(* PLC project ammonium-nitrates, Generated TextualNotationConverter 1.0 *)
(* stored: creationDateTime 2025-07-30T12:00:00, modificationDateTime 2025-01-30T12:00:00 *)

FUNCTION_BLOCK ANALOG_IN
  VAR_INPUT
    Name : STRING;
    Description : STRING;
    Raw_Signal : REAL;
    PV_High : REAL;
    PV_Low : REAL;
    Scaling_Slope : REAL;
    Scaling_Offset : REAL;
    Alarm_Enable : BOOL;
  END_VAR
  VAR_OUTPUT
    PV : REAL;
    High_Alarm : BOOL;
    Low_Alarm : BOOL;
    General_Fault : BOOL;
  END_VAR

            
          
END_FUNCTION_BLOCK

FUNCTION_BLOCK BOOL_IN
  VAR_INPUT
    Name : STRING;
    Description : STRING;
    Bool_In : BOOL;
    Alarm_OnTrue : BOOL;
    Alarm_OnFalse : BOOL;
    Latch_Enable : BOOL;
    Reset_Latch : BOOL;
  END_VAR
  VAR_OUTPUT
    Bool_Out : BOOL;
    Alarm_Active : BOOL;
    Latched_Status : BOOL;
  END_VAR

            
          
END_FUNCTION_BLOCK

FUNCTION_BLOCK PID_BASIC
  VAR_INPUT
    Name : STRING;
    Description : STRING;
    AUTO : BOOL;
    PV : REAL;
    SP : REAL;
    MV_MIN : REAL;
    MV_MAX : REAL;
    X0 : REAL;
    KP : REAL;
    TR : REAL;
    TD : REAL;
    PV_High : REAL;
    PV_Low : REAL;
    Deviation_Limit : REAL;
    Inhibit : BOOL;
  END_VAR
  VAR_OUTPUT
    PV_High_Alarm : BOOL;
    PV_Low_Alarm : BOOL;
    Deviation_Alarm : BOOL;
    XOUT : REAL;
  END_VAR

            
          
END_FUNCTION_BLOCK

FUNCTION_BLOCK RATIO_CONTROL
  VAR_INPUT
    Name : STRING;
    Description : STRING;
    Auto : BOOL;
    PrimaryPV : REAL;
    SecondaryPV : REAL;
    RatioSP : REAL;
    Bias : REAL;
    TrimKp : REAL;
    TrimTi : STRING;
    MV_MIN : REAL;
    MV_MAX : REAL;
    ManOut : REAL;
    Inhibit : BOOL;
  END_VAR
  VAR_OUTPUT
    SlaveSP : REAL;
    ActiveRatio : REAL;
    RatioErr : REAL;
  END_VAR

            
          
END_FUNCTION_BLOCK

FUNCTION_BLOCK VALVE_ELECTRIC
  VAR_INPUT
    Name : STRING;
    Description : STRING;
    Control_Signal : REAL;
    Manual_Mode : BOOL;
    Manual_Position : REAL;
    Open_Limit : REAL;
    Close_Limit : REAL;
    Timeout : STRING;
    Inhibit : BOOL;
  END_VAR
  VAR_OUTPUT
    Valve_Position : REAL;
    Feedback_Pos : REAL;
    Valve_Moving : BOOL;
    Position_Error : BOOL;
    Alarm : BOOL;
  END_VAR

            
          
END_FUNCTION_BLOCK

PROGRAM Section2
  VAR
    FIC102_AcidFlow_SP_FromRatio : REAL;
    FV102_ValveCmd_Pct : REAL;
    FV101_ValveCmd_Pct : REAL;
    FT101_AmmoniaFlow_PV : REAL;
  END_VAR
  VAR
    FT-101 : ANALOG_IN;
    FT-102 : ANALOG_IN;
    LT-104 : ANALOG_IN;
    PH-105 : ANALOG_IN;
    FIC-101 : PID_BASIC;
    FIC-102 : PID_BASIC;
    TIC-103 : PID_BASIC;
    FFIC-102 : RATIO_CONTROL;
    FV-101 : VALVE_ELECTRIC;
    FV-102 : VALVE_ELECTRIC;
    VS-107 : BOOL_IN;
  END_VAR
  VAR  (* added by the conversion: wires and edge detectors of the diagram *)
    _OR1_OUT : BOOL;
  END_VAR

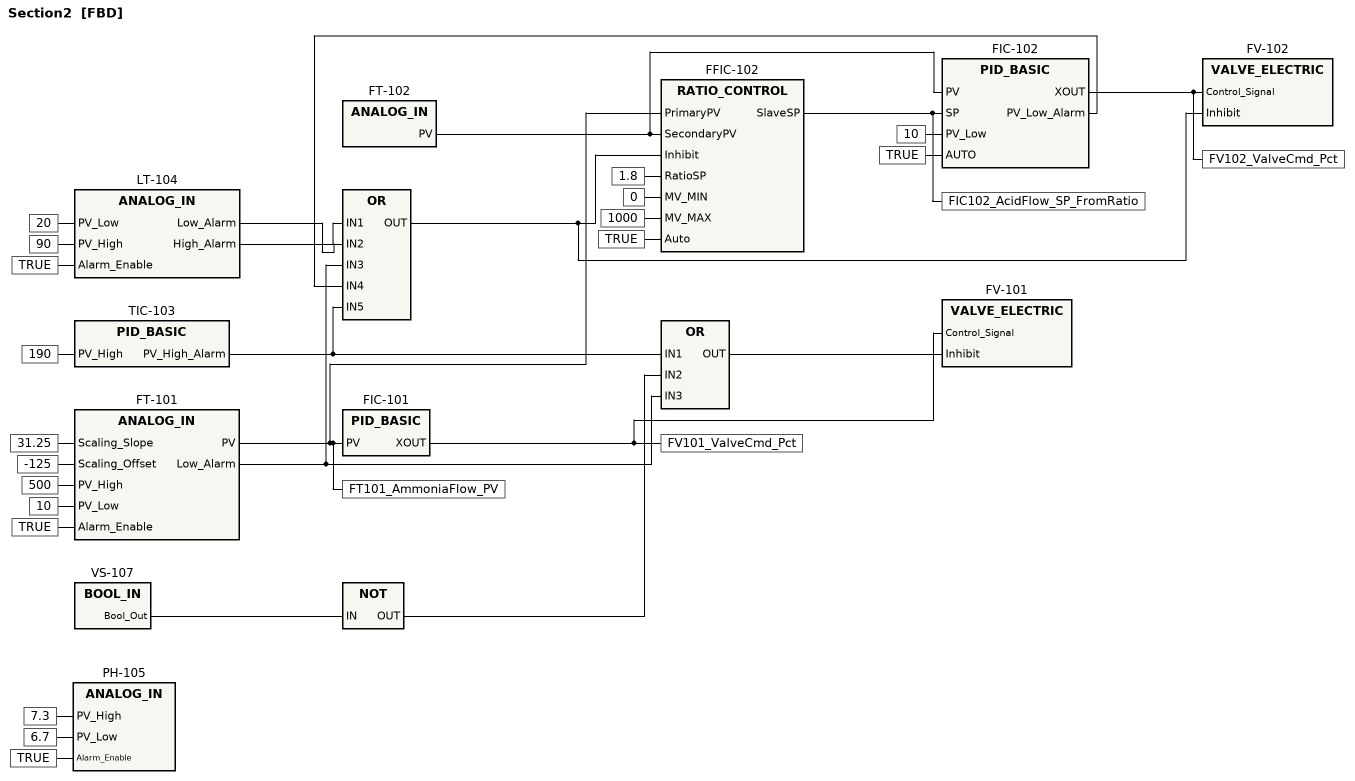
(* FBD diagram, written out as Structured Text *)
FT-101(Scaling_Slope := 31.25, Scaling_Offset := -125, PV_High := 500, PV_Low := 10, Alarm_Enable := TRUE);
FT-102();
LT-104(PV_Low := 20, PV_High := 90, Alarm_Enable := TRUE);
FIC-102(PV := FT-102.PV, SP := FFIC-102.SlaveSP, PV_Low := 10, AUTO := TRUE);
TIC-103(PV_High := 190);
_OR1_OUT := LT-104.High_Alarm OR LT-104.Low_Alarm OR FT-101.Low_Alarm OR FIC-102.PV_Low_Alarm OR TIC-103.PV_High_Alarm;
FFIC-102(PrimaryPV := FT-101.PV, SecondaryPV := FT-102.PV, Inhibit := _OR1_OUT, RatioSP := 1.8, MV_MIN := 0, MV_MAX := 1000, Auto := TRUE);
FIC102_AcidFlow_SP_FromRatio := FFIC-102.SlaveSP;
FT101_AmmoniaFlow_PV := FT-101.PV;
FIC-101(PV := FT-101.PV);
FV101_ValveCmd_Pct := FIC-101.XOUT;
FV102_ValveCmd_Pct := FIC-102.XOUT;
VS-107();
PH-105(PV_High := 7.3, PV_Low := 6.7, Alarm_Enable := TRUE);
FV-101(Control_Signal := FIC-101.XOUT, Inhibit := TIC-103.PV_High_Alarm OR NOT VS-107.Bool_Out OR FT-101.Low_Alarm);
FV-102(Control_Signal := FIC-102.XOUT, Inhibit := _OR1_OUT);
END_PROGRAM

FUNCTION_BLOCK DIGITAL_IN
  VAR_INPUT
    Name : STRING;
    Description : STRING;
    DI_Raw : BOOL;
    DebounceTime : STRING;
    EnableAlarm : BOOL;
  END_VAR
  VAR_OUTPUT
    DI_Out : BOOL;
    Fault_State : BOOL;
  END_VAR

            
          
END_FUNCTION_BLOCK

FUNCTION_BLOCK DUTY_STANDBY
  VAR_INPUT
    Name : STRING;
    Description : STRING;
    Enable : BOOL;
    StartRequest : BOOL;
    AlternateEnable : BOOL;
    ForcePumpA : BOOL;
    ForcePumpB : BOOL;
    DutyElapsed : BOOL;
    MinRunElapsed : BOOL;
    SwitchoverDelayElapsed : BOOL;
    StartTimeoutElapsed : BOOL;
    PumpA_RunFB : BOOL;
    PumpB_RunFB : BOOL;
    PumpA_Fault : BOOL;
    PumpB_Fault : BOOL;
    Reset : BOOL;
    Inhibit : BOOL;
  END_VAR
  VAR_OUTPUT
    CmdPumpA : BOOL;
    CmdPumpB : BOOL;
    ActiveIsA : BOOL;
    SwitchedDueToDuty : BOOL;
    SwitchedDueToFailure : BOOL;
    Alarm_FailedStart_A : BOOL;
    Alarm_FailedStart_B : BOOL;
    Alarm_NoAvailablePump : BOOL;
  END_VAR

            
          
END_FUNCTION_BLOCK

FUNCTION_BLOCK MOTOR_2SPD
  VAR_INPUT
    Name : STRING;
    Description : STRING;
    Start_Cmd : BOOL;
    Stop_Cmd : BOOL;
    Speed_High_Cmd : BOOL;
    Speed_Low_Cmd : BOOL;
    Inhibit : BOOL;
  END_VAR
  VAR_OUTPUT
    Motor_Start_Out : BOOL;
    FB_Running : BOOL;
    FB_Trip : BOOL;
    FB_HighSpeed : BOOL;
    FB_LowSpeed : BOOL;
    Alarm_Speed_Error : BOOL;
  END_VAR

            
          
END_FUNCTION_BLOCK

FUNCTION_BLOCK MOTOR_ON_OFF
  VAR_INPUT
    Name : STRING;
    Description : STRING;
    Start_Cmd : BOOL;
    Stop_Cmd : BOOL;
    Start_Delay : STRING;
    MinRunTime : STRING;
    Inhibit : BOOL;
  END_VAR
  VAR_OUTPUT
    Motor_Start_Out : BOOL;
    FB_Running : BOOL;
    FB_Trip : BOOL;
    Alarm_Start_Fail : BOOL;
    Alarm_Stop_Fail : BOOL;
  END_VAR

            
          
END_FUNCTION_BLOCK

FUNCTION_BLOCK MOTOR_VSD
  VAR_INPUT
    Name : STRING;
    Description : STRING;
    Start_Cmd : BOOL;
    Stop_Cmd : BOOL;
    Speed_SP : REAL;
    Accel_Ramp : STRING;
    Decel_Ramp : STRING;
    Inhibit : BOOL;
  END_VAR
  VAR_OUTPUT
    Speed_Out : REAL;
    FB_Running : BOOL;
    FB_Fault : BOOL;
    FB_Ready : BOOL;
    FB_ActualSpeed : REAL;
    Alarm_Speed_Deviation : BOOL;
    Alarm_Comm_Fail : BOOL;
  END_VAR

            
          
END_FUNCTION_BLOCK

FUNCTION_BLOCK SPLIT_RANGE
  VAR_INPUT
    Name : STRING;
    Description : STRING;
    IN : REAL;
    Split_Point : REAL;
    Output1_Start : REAL;
    Output1_End : REAL;
    Output2_Start : REAL;
    Output2_End : REAL;
  END_VAR
  VAR_OUTPUT
    OUT1 : REAL;
    OUT2 : REAL;
  END_VAR

            
          
END_FUNCTION_BLOCK

FUNCTION_BLOCK VALVE_ON_OFF
  VAR_INPUT
    Name : STRING;
    Description : STRING;
    Open_Cmd : BOOL;
    Close_Cmd : BOOL;
    Timeout : STRING;
    Inhibit : BOOL;
  END_VAR
  VAR_OUTPUT
    FB_Opened : BOOL;
    FB_Closed : BOOL;
    Valve_Open_Out : BOOL;
    Valve_Close_Out : BOOL;
    Alarm_Position_Error : BOOL;
    Alarm_General : BOOL;
  END_VAR

            
          
END_FUNCTION_BLOCK

FUNCTION_BLOCK VOTING_ANALOG
  VAR_INPUT
    Name : STRING;
    Description : STRING;
    Input1 : REAL;
    Input2 : REAL;
    Input3 : REAL;
    Deviation_Limit : REAL;
    Voting_Scheme : STRING;
    EnableAlarm : BOOL;
    Inhibit : BOOL;
  END_VAR
  VAR_OUTPUT
    Voted_Output : REAL;
    Sensor1_Fault : BOOL;
    Sensor2_Fault : BOOL;
    Sensor3_Fault : BOOL;
    Alarm_Voting_Error : BOOL;
    Healthy_Sensors_Count : INT;
  END_VAR

            
          
END_FUNCTION_BLOCK

PROGRAM Section3
  VAR
    TIC201_RSP_to_FIC102 : REAL;
    FIC102_MV_to_FV102 : REAL;
    TT103_MeltTemp_PV : REAL;
    TT104_SteamTemp_PV : REAL;
    PT203_VacuumPressure_PV : REAL;
  END_VAR
  VAR
    TIC-201 : PID_BASIC;
    FIC-102 : PID_BASIC;
    TT-103 : ANALOG_IN;
    TT-104 : ANALOG_IN;
    PT-203 : ANALOG_IN;
    FV-102 : VALVE_ELECTRIC;
    PV-106 : VALVE_ELECTRIC;
    XV-101 : VALVE_ON_OFF;
    P-205 : MOTOR_ON_OFF;
    HS-204 : BOOL_IN;
    VS-206 : DIGITAL_IN;
  END_VAR
  VAR  (* added by the conversion: wires and edge detectors of the diagram *)
    _OR37_OUT : BOOL;
    _OR39_OUT : BOOL;
    _OR43_OUT : BOOL;
    _OR38_OUT : BOOL;
    _NOT40_OUT : BOOL;
  END_VAR

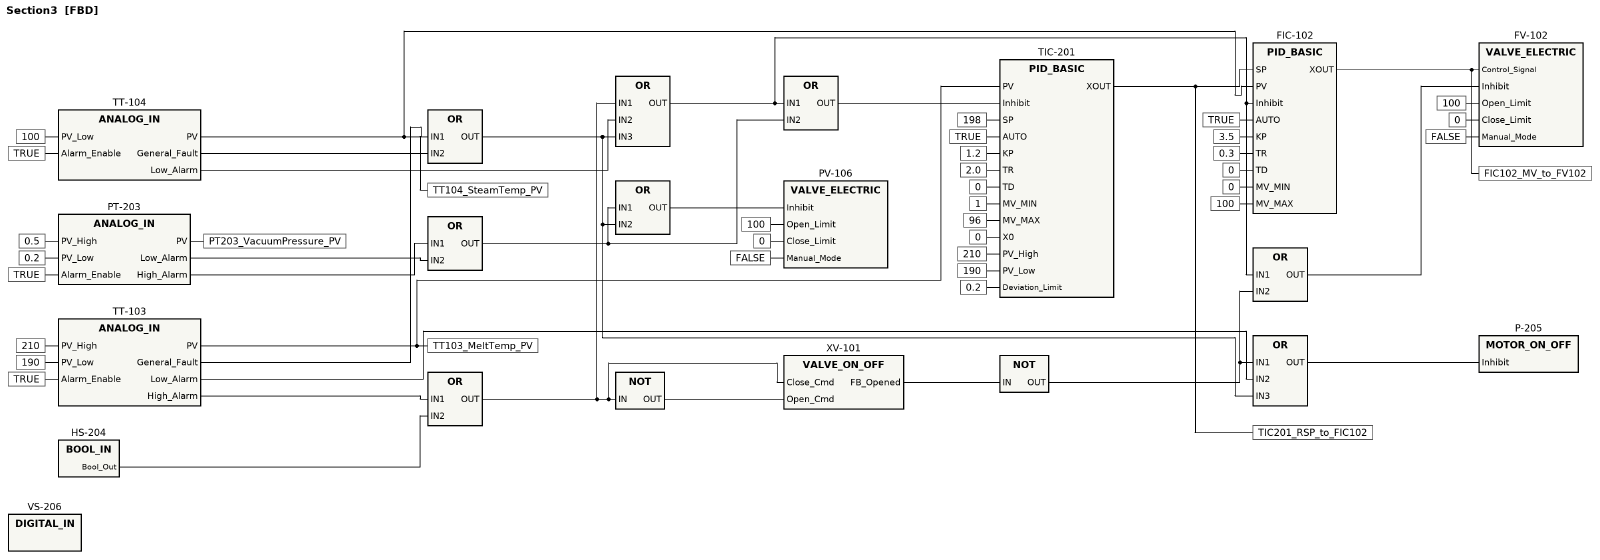
(* FBD diagram, written out as Structured Text *)
TT-103(PV_High := 210, PV_Low := 190, Alarm_Enable := TRUE);
HS-204();
_OR37_OUT := TT-103.High_Alarm OR HS-204.Bool_Out;
TT-104(PV_Low := 100, Alarm_Enable := TRUE);
_OR39_OUT := TT-103.General_Fault OR TT-104.General_Fault;
_OR43_OUT := _OR37_OUT OR TT-104.Low_Alarm OR _OR39_OUT;
PT-203(PV_High := 0.5, PV_Low := 0.2, Alarm_Enable := TRUE);
_OR38_OUT := PT-203.High_Alarm OR PT-203.Low_Alarm;
TIC-201(PV := TT-103.PV, Inhibit := _OR43_OUT OR _OR38_OUT, SP := 198, AUTO := TRUE, KP := 1.2, TR := 2.0, TD := 0, MV_MIN := 1, MV_MAX := 96, X0 := 0, PV_High := 210, PV_Low := 190, Deviation_Limit := 0.2);
FIC-102(SP := TIC-201.XOUT, PV := TT-104.PV, Inhibit := _OR43_OUT, AUTO := TRUE, KP := 3.5, TR := 0.3, TD := 0, MV_MIN := 0, MV_MAX := 100);
FIC102_MV_to_FV102 := FIC-102.XOUT;
PT203_VacuumPressure_PV := PT-203.PV;
TIC201_RSP_to_FIC102 := TIC-201.XOUT;
TT103_MeltTemp_PV := TT-103.PV;
TT104_SteamTemp_PV := TT-104.PV;
XV-101(Close_Cmd := _OR37_OUT, Open_Cmd := NOT _OR37_OUT);
_NOT40_OUT := NOT XV-101.FB_Opened;
FV-102(Control_Signal := FIC-102.XOUT, Inhibit := _OR43_OUT OR _NOT40_OUT, Open_Limit := 100, Close_Limit := 0, Manual_Mode := FALSE);
PV-106(Inhibit := _OR38_OUT OR _OR39_OUT, Open_Limit := 100, Close_Limit := 0, Manual_Mode := FALSE);
P-205(Inhibit := _NOT40_OUT OR TT-103.Low_Alarm OR _OR39_OUT);
VS-206();
END_PROGRAM

PROGRAM Section4
  VAR
    TIC_302_RSP_to_FIC_301 : REAL;
    FIC_301_MeltFlow_ControlSignal_to_FV_301 : REAL;
    GR306_Collecting : BOOL;
  END_VAR
  VAR
    AT-303 : ANALOG_IN;
    FIC-301 : PID_BASIC;
    FT-301 : ANALOG_IN;
    FV-301 : VALVE_ELECTRIC;
    GR-306 : BOOL_IN;
    PR-305 : ANALOG_IN;
    RTD-302 : ANALOG_IN;
    TIC-302 : PID_BASIC;
    VS-304 : ANALOG_IN;
  END_VAR
  VAR  (* added by the conversion: wires and edge detectors of the diagram *)
    _OR97_OUT : BOOL;
  END_VAR

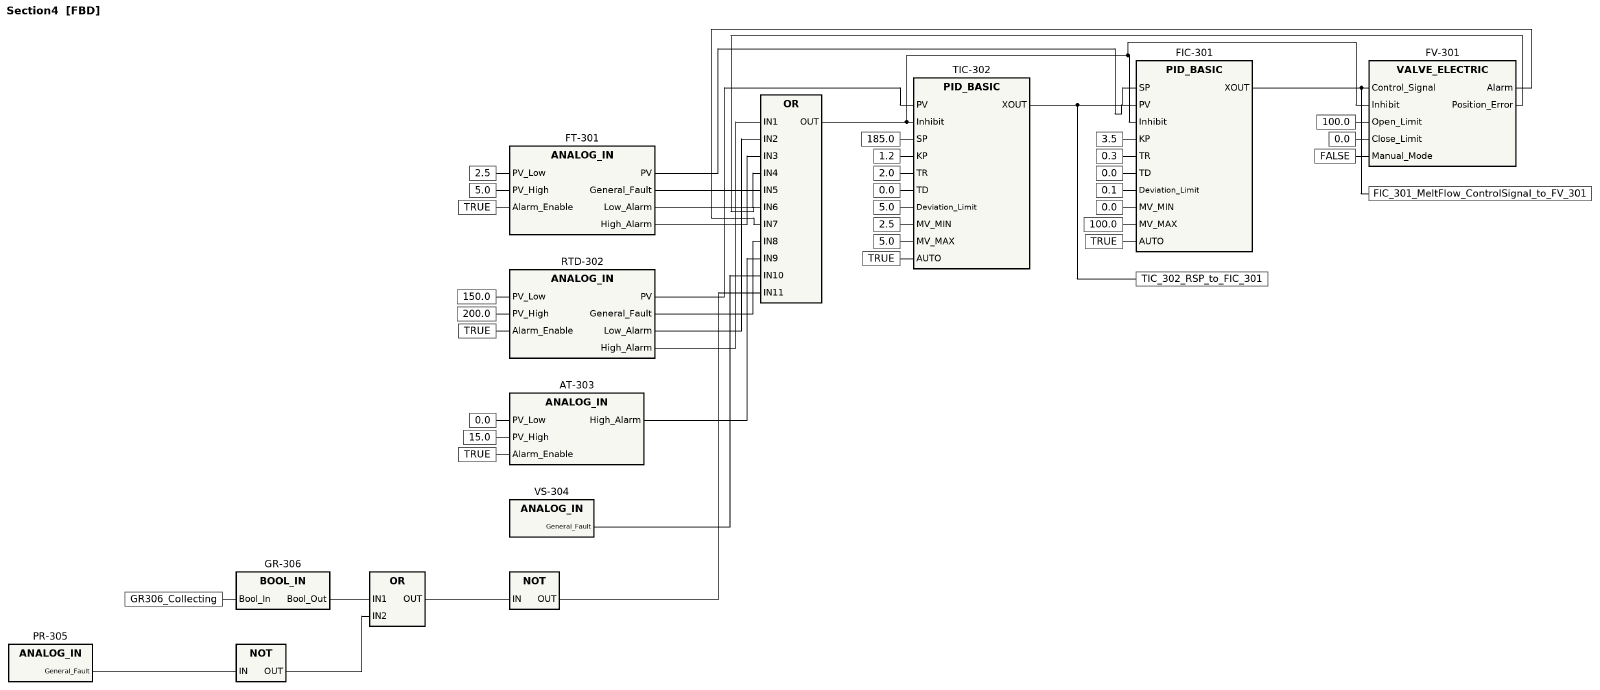
(* FBD diagram, written out as Structured Text *)
RTD-302(PV_Low := 150.0, PV_High := 200.0, Alarm_Enable := TRUE);
FT-301(PV_Low := 2.5, PV_High := 5.0, Alarm_Enable := TRUE);
FV-301(Control_Signal := FIC-301.XOUT, Inhibit := _OR97_OUT, Open_Limit := 100.0, Close_Limit := 0.0, Manual_Mode := FALSE);
AT-303(PV_Low := 0.0, PV_High := 15.0, Alarm_Enable := TRUE);
VS-304();
GR-306(Bool_In := GR306_Collecting);
PR-305();
_OR97_OUT := RTD-302.High_Alarm OR RTD-302.Low_Alarm OR FT-301.High_Alarm OR FT-301.Low_Alarm OR FT-301.General_Fault OR FV-301.Position_Error OR FV-301.Alarm OR RTD-302.General_Fault OR AT-303.High_Alarm OR VS-304.General_Fault OR NOT (GR-306.Bool_Out OR NOT PR-305.General_Fault);
TIC-302(PV := RTD-302.PV, Inhibit := _OR97_OUT, SP := 185.0, KP := 1.2, TR := 2.0, TD := 0.0, Deviation_Limit := 5.0, MV_MIN := 2.5, MV_MAX := 5.0, AUTO := TRUE);
FIC-301(SP := TIC-302.XOUT, PV := FT-301.PV, Inhibit := _OR97_OUT, KP := 3.5, TR := 0.3, TD := 0.0, Deviation_Limit := 0.1, MV_MIN := 0.0, MV_MAX := 100.0, AUTO := TRUE);
FIC_301_MeltFlow_ControlSignal_to_FV_301 := FIC-301.XOUT;
TIC_302_RSP_to_FIC_301 := TIC-302.XOUT;
END_PROGRAM

PROGRAM Section5
  VAR
    TT_401_Temp_PV_C : REAL;
    FT_402_Flow_PV_LPM : REAL;
    FV_402_Valve_Position_Pct : REAL;
    MP_405_Motor_Start_Out : BOOL;
  END_VAR
  VAR
    TIC-401 : PID_BASIC;
    FIC-402 : PID_BASIC;
    TT-401 : ANALOG_IN;
    FT-402 : ANALOG_IN;
    FV-402 : VALVE_ELECTRIC;
    MP-405 : MOTOR_ON_OFF;
    PS-403 : BOOL_IN;
    PSA-404 : DIGITAL_IN;
  END_VAR
  VAR  (* added by the conversion: wires and edge detectors of the diagram *)
    _OR137_OUT : BOOL;
    _OR138_OUT : BOOL;
  END_VAR

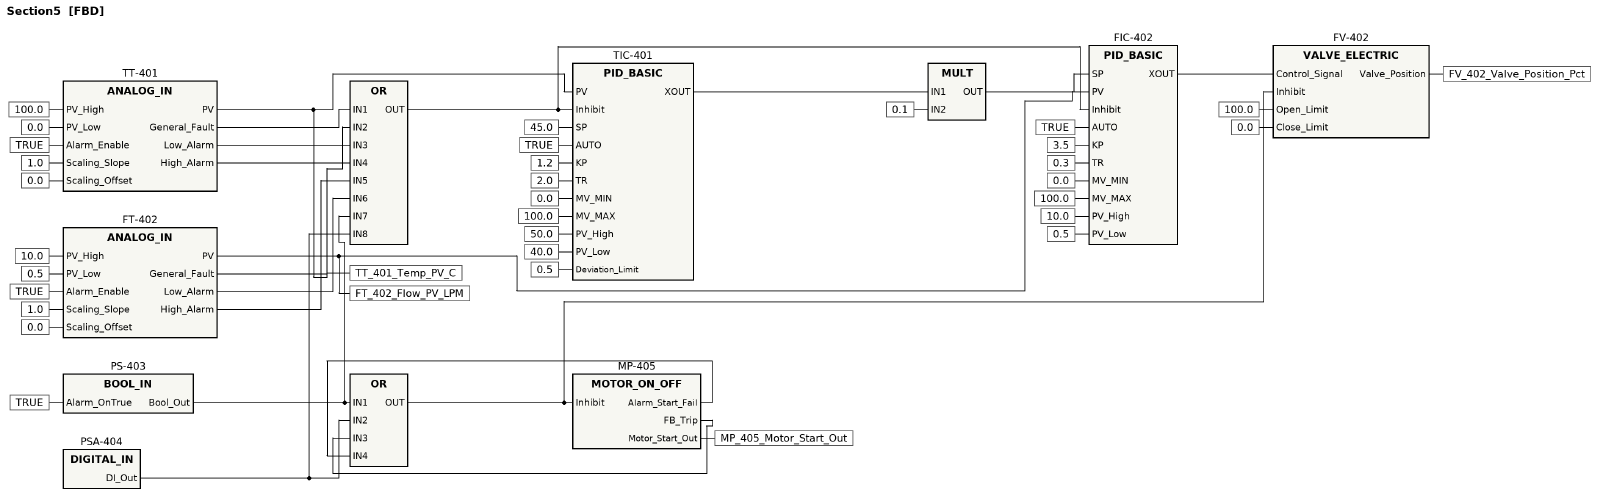
(* FBD diagram, written out as Structured Text *)
FT-402(PV_High := 10.0, PV_Low := 0.5, Alarm_Enable := TRUE, Scaling_Slope := 1.0, Scaling_Offset := 0.0);
FT_402_Flow_PV_LPM := FT-402.PV;
TT-401(PV_High := 100.0, PV_Low := 0.0, Alarm_Enable := TRUE, Scaling_Slope := 1.0, Scaling_Offset := 0.0);
PS-403(Alarm_OnTrue := TRUE);
PSA-404();
_OR137_OUT := TT-401.General_Fault OR TT-401.High_Alarm OR TT-401.Low_Alarm OR FT-402.General_Fault OR FT-402.High_Alarm OR FT-402.Low_Alarm OR PS-403.Bool_Out OR PSA-404.DI_Out;
TIC-401(PV := TT-401.PV, Inhibit := _OR137_OUT, SP := 45.0, AUTO := TRUE, KP := 1.2, TR := 2.0, MV_MIN := 0.0, MV_MAX := 100.0, PV_High := 50.0, PV_Low := 40.0, Deviation_Limit := 0.5);
FIC-402(SP := MULT(TIC-401.XOUT, 0.1), PV := FT-402.PV, Inhibit := _OR137_OUT, AUTO := TRUE, KP := 3.5, TR := 0.3, MV_MIN := 0.0, MV_MAX := 100.0, PV_High := 10.0, PV_Low := 0.5);
MP-405(Inhibit := _OR138_OUT);
_OR138_OUT := PS-403.Bool_Out OR PSA-404.DI_Out OR MP-405.FB_Trip OR MP-405.Alarm_Start_Fail;
FV-402(Control_Signal := FIC-402.XOUT, Inhibit := _OR138_OUT, Open_Limit := 100.0, Close_Limit := 0.0);
FV_402_Valve_Position_Pct := FV-402.Valve_Position;
MP_405_Motor_Start_Out := MP-405.Motor_Start_Out;
TT_401_Temp_PV_C := TT-401.PV;
END_PROGRAM

PROGRAM Section6
  VAR
    WB505_FlowRate_PV : REAL;
    LT501_SiloLevel_PV : REAL;
    SC504_FlowSP_Calc : REAL;
    SC504_SpeedCmd : REAL;
    SC504_Flow_PV : REAL;
    AP503_AerationActive_Status : BOOL;
    PRV502_Closed_Status : BOOL;
  END_VAR
  VAR
    LT-501 : ANALOG_IN;
    WB-505 : ANALOG_IN;
    RIC-506 : RATIO_CONTROL;
    FIC-507 : PID_BASIC;
    SC-504 : MOTOR_VSD;
    AP-503 : BOOL_IN;
    PRV-502 : BOOL_IN;
  END_VAR
  VAR  (* added by the conversion: wires and edge detectors of the diagram *)
    _MULT185_OUT : ANY;
    _OR184_OUT : BOOL;
  END_VAR

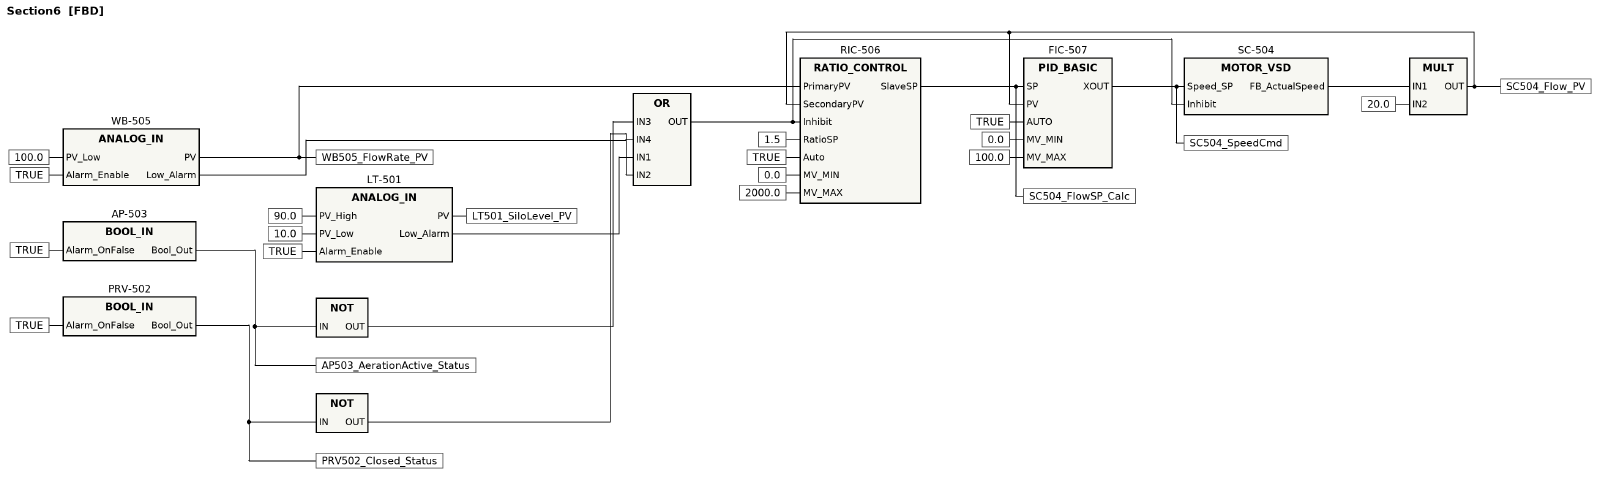
(* FBD diagram, written out as Structured Text *)
AP-503(Alarm_OnFalse := TRUE);
AP503_AerationActive_Status := AP-503.Bool_Out;
LT-501(PV_High := 90.0, PV_Low := 10.0, Alarm_Enable := TRUE);
LT501_SiloLevel_PV := LT-501.PV;
PRV-502(Alarm_OnFalse := TRUE);
PRV502_Closed_Status := PRV-502.Bool_Out;
WB-505(PV_Low := 100.0, Alarm_Enable := TRUE);
FIC-507(SP := RIC-506.SlaveSP, PV := _MULT185_OUT, AUTO := TRUE, MV_MIN := 0.0, MV_MAX := 100.0);
_OR184_OUT := NOT AP-503.Bool_Out OR NOT PRV-502.Bool_Out OR LT-501.Low_Alarm OR WB-505.Low_Alarm;
SC-504(Speed_SP := FIC-507.XOUT, Inhibit := _OR184_OUT);
_MULT185_OUT := MULT(SC-504.FB_ActualSpeed, 20.0);
RIC-506(PrimaryPV := WB-505.PV, SecondaryPV := _MULT185_OUT, Inhibit := _OR184_OUT, RatioSP := 1.5, Auto := TRUE, MV_MIN := 0.0, MV_MAX := 2000.0);
SC504_FlowSP_Calc := RIC-506.SlaveSP;
SC504_Flow_PV := _MULT185_OUT;
SC504_SpeedCmd := FIC-507.XOUT;
WB505_FlowRate_PV := WB-505.PV;
END_PROGRAM

CONFIGURATION Config0
  RESOURCE Res0 ON PLC
    TASK task0(INTERVAL := T#20ms, PRIORITY := 0);
    PROGRAM instance0 WITH task0 : Section2;
    PROGRAM instance_1 WITH task0 : Section3;
    PROGRAM instance_2 WITH task0 : Section4;
    PROGRAM instance_3 WITH task0 : Section5;
    PROGRAM instance_4 WITH task0 : Section6;
  END_RESOURCE
END_CONFIGURATION
